{attribute 'GeneratedUsingTerminal: AT2040-0250-0023'}
{attribute addProperty BoxType "AT2040-0250-0023"}
{attribute addProperty Id "A_0106_AT2026_5250_0019_AT2026_5250AT2026_01D6DEDF80"}
{attribute addProperty CRC "1369845472"}
{attribute addProperty Size "80"}
TYPE A_0038_AT2040_0250_0023_51A62EE0 EXTENDS AT2040_86175B41 :
STRUCT
	{attribute addProperty Name "A_0106_AT2026_5250_0019_AT2026_5250"}
	{attribute addProperty PreviousPort "A_0038(AT2040-0250-0023) : B"}
	A_0106_AT2026_5250_0019_AT2026_5250 : AT2026_01D6DEDF;
END_STRUCT
END_TYPE

(* stored: Version 1.2.0.0, ProductVersion 3.1.4024.9
   DUT A_0038_AT2040_0250_0023_51A62EE0: Id {7503e719-5e37-42c0-a28f-6be08e845870} *)
